TYPE EL2044_Diag :
STRUCT
	{attribute addProperty Name "Channel 1"}
	_1 AT %I* : DIGDiagInput;
	{attribute addProperty Name "Channel 2"}
	_2 AT %I* : DIGDiagInput;
	{attribute addProperty Name "Channel 3"}
	_3 AT %I* : DIGDiagInput;
	{attribute addProperty Name "Channel 4"}
	_4 AT %I* : DIGDiagInput;
END_STRUCT
END_TYPE

(* stored: Version 1.1.0.1, ProductVersion 3.1.4024.9
   DUT EL2044_Diag: Id {92a21d7f-c20d-016b-0bd8-3ca44b818569} *)
